Staubli VAL3: SocketMove.pjx

--- SocketMove.pjx ---
Parameters version=s7.8.3 stackSize=5000 millimeterUnit=true
Program file=Safety.pgx
Program file=SpeedFilter.pgx
Program file=SplitJoint.pgx
Program file=SplitMoveC.pgx
Program file=SplitMoveJ.pgx
Program file=SplitMoveL.pgx
Program file=SplitNumS.pgx
Program file=SplitPresetLine.pgx
Program file=SplitString.pgx
Program file=SplitTrsf.pgx
Program file=start.pgx
Program file=stop.pgx
Data file=SocketMove.dtx

--- SocketMove.dtx ---
mdesc mNomSpeed
string sGetStr
sio sS = {link=Socket\ss}
string sBuff
trsf trTrsf
trsf trPara
bool bRes
mdesc mRun
pointRx pPrun = {fatherId=world[0]}
tool tTool = {z=100, fatherId=flange[0], ioLink=valve1}
jointRx jrun
pointRx pPMovec = {fatherId=world[0]}
pointRx pCurrent = {fatherId=world[0]}
trsf trSafety = {x=924.6, y=357.15, z=-147.43, ry=-180, rz=-1.37}
bool bOverRun
num nRobotSpeed

--- start.pgx ---
program start()
begin

  cls()
  title("通过socket传送数据来实现运动")
  //初始化
  taskCreateSync  "safetyCheck",0.008,bOverRun,Safety()
  clearBuffer(sS)
  sGetStr=""
  resetMotion()
  wait(isPowered())


  //循环语句
  while isPowered()

    sGetStr=sS
    if find(sGetStr,"MOVEL")>=0
      call SplitMoveL(sGetStr,trTrsf,trPara,true,bRes)
      if !bRes
        popUpMsg("数据不对")
        return
      endIf
      call SpeedFilter(trPara,mRun)
      link(pPrun,world)
      pPrun.trsf=trTrsf
      movel(pPrun,tTool,mRun)
    endIf

    if find(sGetStr,"MOVEJ")>=0
      call SplitMoveJ(sGetStr,jrun,trPara,false,bRes)
      if !bRes
        popUpMsg("数据不对")
        return
      endIf
      call SpeedFilter(trPara,mRun)
      movej(jrun,tTool,mRun)
    endIf


    if find(sGetStr,"MOVEC")>=0
      call SplitMoveC(sGetStr,pPMovec.trsf,trTrsf,trPara,bRes)
      if !bRes
        popUpMsg("数据不对")
        return
      endIf
      call SpeedFilter(trPara,mRun)
      link(pPrun,world)
      pPrun.trsf=trTrsf
      link(pPMovec,world)
      movec(pPMovec,pPrun,tTool,mRun)
    endIf

    //进行握手
    if sGetStr!=""
      sS="success"
    endIf


  endWhile
  resetMotion()



end

--- Safety.pgx ---
program Safety()
begin

  //同步任务来实现安全检测
  while true
    //获取速度
    nRobotSpeed=getSpeed(tTool)


    //判断位置是否超过安全区域
    pCurrent=here(tTool,world)
    if distance(pCurrent.trsf,trSafety)>200
      if isPowered()
        popUpMsg("超过安全限制")
        disablePower()
      endIf
    endIf
    delay(0)
  endWhile


end

--- SpeedFilter.pgx ---
public program SpeedFilter(trsf x_tr, mdesc& x_mDest)
  local num l_nDist
begin

 // DataBase:nSpeedPercent=min(max(0.001,DataBase:nSpeedPercent),100)



  //调试系数
  //l_nPercent=2
  //








  x_mDest.decel=x_mDest.accel=max(x_tr.rx,0.1)*1
  x_mDest.blend=Cartesian
   // x_mDest.blend=joint
  x_mDest.reach=x_mDest.leave=max(x_tr.ry,0)
  x_mDest.tvel=max(x_tr.z,0.1)*1
  x_mDest.vel=100
  x_mDest.rvel=99999


end

--- SplitMoveC.pgx ---
public program SplitMoveC(string x_sSLine, trsf& x_tr1, trsf& x_tr2, trsf& x_trP, bool& x_bRes)
  local string l_sChar[2]
  local num l_nData[25]
begin
  x_bRes=false

  if x_sSLine==""
    return
  endIf

  x_sSLine=right(x_sSLine,len(x_sSLine)-len("MOVEC="))

  //解析每一行
  l_sChar[0]=","
  l_sChar[1]="/"

  call SplitNumS(x_sSLine,l_nData,l_sChar,x_bRes)

  if !x_bRes
    return
  endIf

  x_tr1.x=l_nData[0]
  x_tr1.y=l_nData[1]
  x_tr1.z=l_nData[2]
  x_tr1.rx=l_nData[3]
  x_tr1.ry=l_nData[4]
  x_tr1.rz=l_nData[5]

  x_tr2.x=l_nData[6]
  x_tr2.y=l_nData[7]
  x_tr2.z=l_nData[8]
  x_tr2.rx=l_nData[9]
  x_tr2.ry=l_nData[10]
  x_tr2.rz=l_nData[11]


  x_trP.x=l_nData[12]
  x_trP.y=l_nData[13]
  x_trP.z=l_nData[14]
  x_trP.rx=l_nData[15]
  x_trP.ry=l_nData[16]
  //x_trP.rz=l_nData[17]




end

--- SplitMoveL.pgx ---
public program SplitMoveL(string x_sSLine, trsf& x_tr1, trsf& x_trP, bool x_bCut, bool& x_bRes)
  local string l_sChar[2]
  local num l_nData[25]
begin
  x_bRes=false

  if x_sSLine==""
    return
  endIf

  x_sSLine=right(x_sSLine,len(x_sSLine)-len("MOVEL="))

  //解析每一行
  l_sChar[0]=","
  l_sChar[1]="/"

  call SplitNumS(x_sSLine,l_nData,l_sChar,x_bRes)

  if !x_bRes
    return
  endIf

  x_tr1.x=l_nData[0]
  x_tr1.y=l_nData[1]
  x_tr1.z=l_nData[2]
  x_tr1.rx=l_nData[3]
  x_tr1.ry=l_nData[4]
  x_tr1.rz=l_nData[5]



  if !x_bCut

    x_trP.z=l_nData[6]
    x_trP.rx=l_nData[7]
  else
    x_trP.x=l_nData[6]
    x_trP.y=l_nData[7]
    x_trP.z=l_nData[8]
    x_trP.rx=l_nData[9]
    x_trP.ry=l_nData[10]
    //x_trP.rz=l_nData[17]

  endIf




end

--- SplitNumS.pgx ---
public program SplitNumS(string x_Source, num& x_Res[], string& x_sChar[], bool& x_bRes)
  local num l_nNum
begin

  call SplitString(x_Source,sBuff,x_sChar,x_bRes)
  if !x_bRes
    return
  endIf



  //把分解的字符串转化为数字量
  for l_nNum=0 to min(size(sBuff)-1,size(x_Res)-1)
    toNum(sBuff[l_nNum],x_Res[l_nNum],x_bRes)
    if !x_bRes
      return
    endIf
  endFor




end

--- SplitPresetLine.pgx ---
public program SplitPresetLine(string x_sLine, num& x_nDest[] (dimensions=2), num x_nFlag, bool& x_bRes)
  local num l_nData[25]
  local num l_nNum
  local num l_nBuff
  local string l_sChar[2]
begin

  x_bRes=false
  if x_sLine==""
    return
  endIf

  // x_sLine=right(x_sLine,len(x_sLine)-find(x_sLine,"=")-1)

  //如果这一行为空
  if x_sLine==""
    x_bRes=true
    return
  endIf


  //解析每一行
  l_sChar[0]=","
  l_sChar[1]=","

  call SplitNumS(x_sLine,l_nData,l_sChar,x_bRes)

  if !x_bRes
    return
  endIf

  l_nBuff=0
  for l_nNum=0 to 4
    //强制对工艺进行设置
    x_nDest[x_nFlag,l_nNum]=max(min(l_nData[l_nBuff],100),0)
    l_nBuff=l_nBuff+1
  endFor












end

--- SplitString.pgx ---
public program SplitString(string x_Source, string& x_sDest[], string& x_sChar[], bool& x_bRes)
  local num l_nResNum
  local string l_sBuff
  local num l_nFlag
  local num l_nBuff
  local num l_nIndex
begin
  //每个函数头格式
  //×××××××××××××××××××××××××××××××××××××××××××××××××
  //函数名：
  //功能：
  //参数含义:
  //使用Addon:
  //作者：
  //备注：x_sDest 只能是全局变量，因为用到了resize函数
  //日期：
  //×××××××××××××××××××××××××××××××××××××××××××××××××

  x_bRes=false
  l_nResNum=0
  resize(x_sDest,1,1)
  x_sDest=""
  if x_Source=="" or x_sChar==""
    return
  endIf

  l_sBuff=x_Source
  while true
    l_nFlag=10000
    //获得最小标志符序号
    for l_nIndex=0 to size(x_sChar)-1 step 1
      l_nBuff=find(l_sBuff,x_sChar[l_nIndex])
      if l_nBuff>=0 and l_nBuff<l_nFlag
        l_nFlag=l_nBuff
      endIf
    endFor


    //里面没有标志符
    if len(l_sBuff)>=1 and l_nFlag==10000
      if l_nResNum!=0
        resize(x_sDest,1,l_nResNum+1)
      endIf
      x_sDest[l_nResNum]=l_sBuff
      x_bRes=true
      return
    endIf

    //字符串为空
    if l_sBuff==""
      x_bRes=true
      return
    endIf


    //分开
    if l_nFlag==0
      l_sBuff=right(l_sBuff,len(l_sBuff)-1)
    else
      if l_nResNum!=0
        resize(x_sDest,1,l_nResNum+1)
      endIf
      x_sDest[l_nResNum]=left(l_sBuff,l_nFlag)
      l_nResNum=l_nResNum+1
      l_sBuff=right(l_sBuff,len(l_sBuff)-l_nFlag-1)
    endIf
  endWhile


end

--- SplitTrsf.pgx ---
public program SplitTrsf(string x_sSLine, string x_sTitle, trsf& x_trTrsf, bool& x_bRes)
  local string l_sChar[2]
  local num l_nData[25]
begin
  x_bRes=false

  if x_sSLine==""
    return
  endIf

  x_sSLine=right(x_sSLine,len(x_sSLine)-len(x_sTitle))

  //解析每一行
  l_sChar[0]=","
  l_sChar[1]=","

  call SplitNumS(x_sSLine,l_nData,l_sChar,x_bRes)

  if !x_bRes
    return
  endIf

  x_trTrsf.x=l_nData[0]
  x_trTrsf.y=l_nData[1]
  x_trTrsf.z=l_nData[2]
  x_trTrsf.rx=l_nData[3]
  x_trTrsf.ry=l_nData[4]
  x_trTrsf.rz=l_nData[5]




end
